TYPE Space :
STRUCT
	Column : SINT;
	Row : SINT;
	PartID : STRING;
	Weight : Weight;
END_STRUCT
END_TYPE

(* stored: Version 1.1.0.1
   DUT Space: Id {b40f7efc-e092-460b-ae27-2957ed094bef} *)
